(* PLC project marvel_shutterplc, Institute of Astronomy Onto 0.0.1 *)
(* stored: creationDateTime 2025-04-10T16:56:59.318796, modificationDateTime 2025-04-10T16:56:59.318796 *)

TYPE DomeShutterApertureStates : (UNKNOWN := 0, FULLY_OPEN := 1, PARTIALLY_OPEN := 2, FULLY_CLOSED := 3, INVALID := 4) BYTE;
END_TYPE

TYPE DomeShutterCommands : (NONE := 0, STOP := 1, CLOSE := 2, OPEN := 3, SET_HUMIDITY_LIMIT := 4, SET_HEARTBEAT_TIMEOUT := 5, SET_DRIVE_LOGIC := 6) BYTE;
END_TYPE

TYPE DomeShutterDriveLogic : (UNKNOWN := 0, EDGE_BASED := 1, LEVEL_BASED := 2) BYTE;
END_TYPE

TYPE DomeShutterMotionStates : (STANDSTILL := 0, OPENING := 1, CLOSING := 2, STOPPING := 3, TIMEOUT_ERROR := 4, RETRY_OPENING := 5, RETRY_CLOSING := 6, UNKNOWN_DRIVE_LOGIC_ERROR := 7) BYTE;
END_TYPE

{attribute 'pack_mode' := '8'}
TYPE DomeShutterDataRead : STRUCT
  {attribute 'TcHmiSymbol.Show'}
  motionState : DomeShutterMotionStates;  (* The motion state, as reported by the shutter PLC *)
  {attribute 'TcHmiSymbol.Show'}
  apertureState : DomeShutterApertureStates;  (* The aperture state, as reported by the shutter PLC *)
  {attribute 'TcHmiSymbol.Show'}
  heartBeatReceived : UDINT;  (* The heartbeat that was last received by the shutter PLC, as reported by the shutter PLC *)
  {attribute 'TcHmiSymbol.Show'}
  lastCommandReceived : DomeShutterCommands;  (* The command that was last received by the shutter PLC, as reported by the shutter PLC *)
  {attribute 'TcHmiSymbol.Show'}
  panelsBottomOpen : BIT;  (* True if the panels are open according to the bottom limit switch *)
  {attribute 'TcHmiSymbol.Show'}
  panelsBottomClosed : BIT;  (* True if the panels are closed according to the bottom limit switch *)
  {attribute 'TcHmiSymbol.Show'}
  panelsTopOpen : BIT;  (* True if the panels are open according to the top limit switch *)
  {attribute 'TcHmiSymbol.Show'}
  panelsTopClosed : BIT;  (* True if the panels are closed according to the top limit switch *)
  {attribute 'TcHmiSymbol.Show'}
  relayOpenActive : BIT;  (* True if the relay to open the shutter is active, False if not *)
  {attribute 'TcHmiSymbol.Show'}
  relayCloseActive : BIT;  (* True if the relay to close the shutter is active, False if not *)
  {attribute 'TcHmiSymbol.Show'}
  bHumidityUnderrange : BIT;  (* True if the humidity sensor is in underrange, False if not *)
  {attribute 'TcHmiSymbol.Show'}
  bHumidityOverrange : BIT;  (* True if the humidity sensor is in overrange, False if not *)
  {attribute 'TcHmiSymbol.Show'}
  bHumidityError : BIT;  (* True if the humidity sensor is in error, False if not *)
  {attribute 'TcHmiSymbol.Show'}
  bTemperatureUnderrange : BIT;  (* True if the temperature sensor is in underrange, False if not *)
  {attribute 'TcHmiSymbol.Show'}
  bTemperatureOverrange : BIT;  (* True if the temperature sensor is in overrange, False if not *)
  {attribute 'TcHmiSymbol.Show'}
  bTemperatureError : BIT;  (* True if the temperature sensor is in error, False if not *)
  {attribute 'TcHmiSymbol.Show'}
  manualOperation : BIT;  (* True if no constraint violation checking is happenening *)
  {attribute 'TcHmiSymbol.Show'}
  heartBeatViolation : BIT;  (* True if there is a missing heartbeat reported by the shutter PLC, False if not *)
  {attribute 'TcHmiSymbol.Show'}
  humidityViolation : BIT;  (* True if there is high humidity reported by the shutter PLC, False if not *)
  {attribute 'TcHmiSymbol.Show'}
  driveLogic : DomeShutterDriveLogic;  (* Determines which logic is used by the shutter drives (edge or level based) *)
  {attribute 'TcHmiSymbol.Show'}
  humidityRawValue : INT;  (* The raw value of the humidity sensor *)
  {attribute 'TcHmiSymbol.Show'}
  temperatureRawValue : INT;  (* The raw value of the temperature sensor *)
  {attribute 'TcHmiSymbol.Show'}
  humidityLimit : INT;  (* Humidity limit (as raw sensor value) above which the dome will close automatically (-1 means turn off) *)
  {attribute 'TcHmiSymbol.Show'}
  heartBeatTimeout : INT;  (* Heartbeat timeout (in seconds) above which the dome will close automatically (-1 means turn off) *)
END_STRUCT;
END_TYPE

{attribute 'pack_mode' := '8'}
TYPE DomeShutterDataWrite : STRUCT
  {attribute 'TcHmiSymbol.Show'}
  heartBeat : UDINT;  (* The heartbeat to send to the shutter PLC *)
  {attribute 'TcHmiSymbol.Show'}
  command : DomeShutterCommands;  (* The command to send to the shutter PLC *)
  {attribute 'TcHmiSymbol.Show'}
  arg : INT;  (* The int16 argument belonging to the command (optional) *)
END_STRUCT;
END_TYPE
